(* CoDeSys 2.3 export: E_MODBUSFUNCTION.EXP *)

(* Data type *)
TYPE E_ModbusFunction : (
	ReadCoils := 1,
	ReadInputStatus := 2,
	ReadRegs := 3,
	ReadInputRegs := 4,
	WriteSingleCoil := 5,
	WriteSingleRegister := 6,
	Diagnostics := 8,
	WriteMultipleCoils := 15,
	WriteRegs := 16
);
END_TYPE
